SUBAPPLICATION Uebung_019c_AX (* Umschalten einer Maske, mit Plug and Socket *)
  (* Standard: 61499-2; Description: Copyright (c) 2026 Meisterschulen am Ostbahnhof This program and the accompanying materials are made available under the terms of the Eclipse Public License 2.0 which is available at https://www.eclipse.org/legal/epl-2.0/ SPDX-License-Identifier: EPL-2.0 *)
  (* Version 1.0, 2026-09-09, Franz Höpfinger, Meisterschulen am Ostbahnhof, initial API and implementation and/or initial documentation *)
  PACKAGE Uebungen;
  IMPORT Uebungen::const::UT::DefaultPool::AlarmMask_A2_medium;
  IMPORT Uebungen::const::UT::DefaultPool::DataMask_M1;
  IMPORT Uebungen::const::UT::DefaultPool::DataMask_M2;
  IMPORT logiBUS::io::DI::logiBUS_DI::Input_I1;
  IMPORT logiBUS::io::DI::logiBUS_DI::Input_I2;
  IMPORT logiBUS::io::DI::logiBUS_DI::Input_I3;
  IMPORT logiBUS::io::DI::logiBUS_DI::Input_I4;
  IMPORT logiBUS::io::DI::logiBUS_DI_Events::BUTTON_SINGLE_CLICK;
  IMPORT logiBUS::io::DQ::logiBUS_DO::Output_Q8;
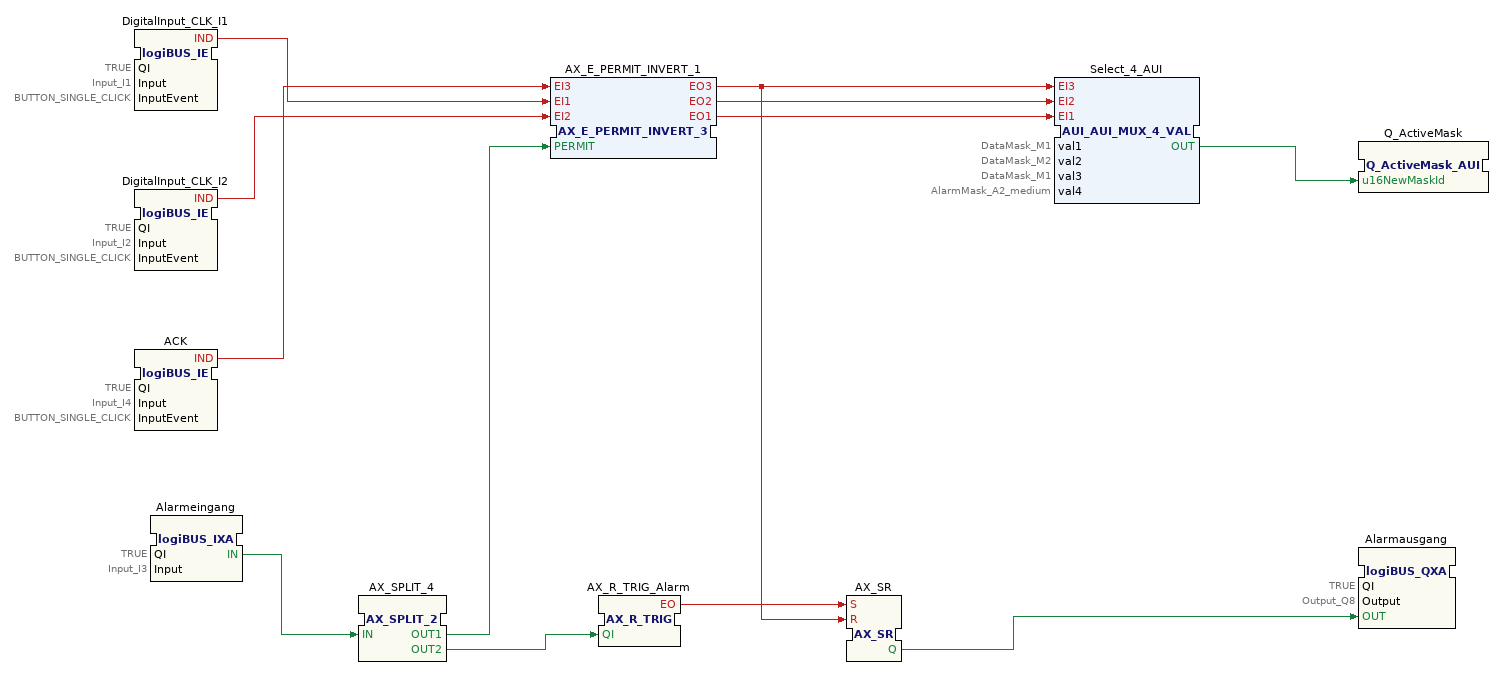
  FBS
    DigitalInput_CLK_I1 : logiBUS::io::DI::logiBUS_IE(QI := TRUE, Input := Input_I1, InputEvent := BUTTON_SINGLE_CLICK);
    DigitalInput_CLK_I2 : logiBUS::io::DI::logiBUS_IE(QI := TRUE, Input := Input_I2, InputEvent := BUTTON_SINGLE_CLICK);
    Q_ActiveMask : isobus::UT::Q::Q_ActiveMask_AUI;
    ACK : logiBUS::io::DI::logiBUS_IE(QI := TRUE, Input := Input_I4, InputEvent := BUTTON_SINGLE_CLICK);
    AX_SR : adapter::events::unidirectional::AX_SR;
    Alarmausgang : logiBUS::io::DQ::logiBUS_QXA(QI := TRUE, Output := Output_Q8);
    Alarmeingang : logiBUS::io::DI::logiBUS_IXA(QI := TRUE, Input := Input_I3);
    AX_R_TRIG_Alarm : adapter::events::unidirectional::AX_R_TRIG;
    AX_SPLIT_4 : adapter::events::unidirectional::AX_SPLIT_2;
  END_FBS
  SUBAPPS
    Select_4_AUI : MyLib::sys::AUI_AUI_MUX_4_VAL(val1 := DataMask_M1, val2 := DataMask_M2, val3 := DataMask_M1, val4 := AlarmMask_A2_medium);
    AX_E_PERMIT_INVERT_1 : MyLib::sys::AX_E_PERMIT_INVERT_3;
  END_SUBAPPS
  EVENT_CONNECTIONS
    AX_R_TRIG_Alarm.EO TO AX_SR.S;
    ACK.IND TO AX_E_PERMIT_INVERT_1.EI3;
    DigitalInput_CLK_I1.IND TO AX_E_PERMIT_INVERT_1.EI1;
    DigitalInput_CLK_I2.IND TO AX_E_PERMIT_INVERT_1.EI2;
    AX_E_PERMIT_INVERT_1.EO3 TO AX_SR.R;
    AX_E_PERMIT_INVERT_1.EO3 TO Select_4_AUI.EI3;
    AX_E_PERMIT_INVERT_1.EO2 TO Select_4_AUI.EI2;
    AX_E_PERMIT_INVERT_1.EO1 TO Select_4_AUI.EI1;
  END_CONNECTIONS
  ADAPTER_CONNECTIONS
    Select_4_AUI.OUT TO Q_ActiveMask.u16NewMaskId;
    AX_SR.Q TO Alarmausgang.OUT;
    Alarmeingang.IN TO AX_SPLIT_4.IN;
    AX_SPLIT_4.OUT1 TO AX_E_PERMIT_INVERT_1.PERMIT;
    AX_SPLIT_4.OUT2 TO AX_R_TRIG_Alarm.QI;
  END_CONNECTIONS
END_SUBAPPLICATION
